// SIMATIC S7-200 project (STEP 7-Micro/WIN), CPU 222 CN REL 02.01

SYMBOL_TABLE 
USS_LOW_V        VD1000
USS_HIGH_V       VD1004
USS_TIME_OUT     VW1008
USS_I_LINE       VW1010
USS_DAT_PTR0     VD1012
USS_ACT_DRV0     VD1016
USS_CUR_DRV0     VD1020
USS_P0           V1024.0
USS_REQ_SNT0     V1024.1
USS_RETRY_P0     VB1025
USS_ERR_CODE     VB1026
USS_CS_D0        VD1027
USS_CS_W0        VW1027
USS_CS_W2        VW1029
USS_CS_B0        VB1027
USS_CS_B1        VB1028
USS_POLL_BUF     VB1031
USS_XMT_0        VB1046
USS_XMT_ADR0     VB1049
USS_X_STWD       VD1056
USS_X_BCC        VB1060
USS_X_DW1        VD1047
USS_X_DW5        VD1051
USS_X_DW9        VD1055
USS_X_DB13       VB1059
USS_RCV_BUF0     VB1061
USS_R_STX        VB1062
USS_R_LGE        VB1063
USS_R_ADR        VB1064
USS_R_STWD       VD1071
USS_R_DW1        VD1062
USS_R_DW5        VD1066
USS_R_DW9        VD1070
USS_R_W13        VW1074
USS_STAT_TAB     VB1076
USS_ADR_P0       VB1396
END_SYMBOL_TABLE

ORGANIZATION_BLOCK 主:OB1
TITLE= 
// 程序注释
// 按 F1 获得帮助及举例程序
//  
// 
BEGIN
Network 1 // 网络题目 (单行)
//  
// 网络注释
//  
// 
LD     SM0.1                 // 首次扫描标志（SM0.1 = 1)
CALL   SBR_0:SBR0            // 调用子程序0，初始化高速输出和HSC0，允许中断
END_ORGANIZATION_BLOCK

SUBROUTINE_BLOCK SBR_0:SBR0
TITLE= 
// 子程序0
//  
// 
BEGIN
Network 1 // 网络题目 (单行)
LD     SM0.0                 // 设置脉冲输出PLS 0的控制字节：允许单段PTO功能，
MOVB   16#8D, SMB67          // 时间基准为ms，可更新脉冲数和周期
R      Q0.0, 1               // 复位脉冲输出Q0.0的映象寄存器
MOVW   +2, SMW68             // 输出脉冲的周期为2ms
MOVD   +12000, SMD72         // 产生12000个脉冲 (共24s)
PLS    0                     // 起动PLS0, 从输出端Q0.0输出脉冲
S      Q0.1, 1               // 在第一段时间（4s）内，Q0.1为1状态
MOVB   16#F8, SMB37          // HSC0初始化，可更新CV、PV和计数方向，加计数
MOVD   +0, SMD38             // HSC0的当前值（CV）清0
MOVD   +2000, SMD42          // HSC0的第一次设定值 (PV) 为2000（延时4s）
HDEF   0, 0                  // 定义HSC0为模式0
ATCH   INT_0:INT0, 12        // HSC0的CV＝PV时，执行中断程序0
ENI                          // 允许全局中断
HSC    0                     // 起动HSC0
END_SUBROUTINE_BLOCK

INTERRUPT_BLOCK INT_0:INT0
TITLE= 
// 中断程序0
// 
// 
BEGIN
Network 1
LD     SM0.0                 // SM0.0总是为ON
R      Q0.1, 1               // 复位Q0.1
S      Q0.2, 1               // 置位Q0.2 
MOVB   16#B0, SMB37          // 重新设置HSC0的控制位，改为减计数
MOVD   +1000, SMD42          // HSC0的第2设定值为1 000
ATCH   INT_1:INT1, 12        // 用中断程序1取代中断程序0，分配给中断事件12 
HSC    0                     // 起动HSC0, 装入新的设定值和计数方向
// 
END_INTERRUPT_BLOCK

INTERRUPT_BLOCK INT_1:INT1
TITLE= 
// 中断程序1
//  
// 
BEGIN
Network 1
LD     SM0.0                 // SM0.0总是为ON
R      Q0.2, 1               // 复位Q0.2 
S      Q0.1, 1               // 置位Q0.1 
MOVB   16#F8, SMB37          // 重新设置HSC0的控制位，改为加计数
MOVD   +0, SMD38             // HSC0的当前值复位（CV=0）
MOVD   +2000, SMD42          // HSC0的设定值（PV)为2 000
ATCH   INT_0:INT0, 12        // 把中断程序0分配给中断事件12 
HSC    0                     // 重新起动HSC 0
// 
END_INTERRUPT_BLOCK
